FUNCTION_BLOCK L2_MedidorTapa_SFC EXTENDS L1_ControllerBase_SFC

VAR_INPUT 							// Sensores y comandos
	dh					: UINT; 	// Detector valor altura 
	// Lectura_Registrada	: BOOL;		// La lectura de la altura ha terminado 	
END_VAR

VAR_OUTPUT							// Actuadores
	L_1: BOOL; 						// Medidor de altura baja
	Leyendo: BOOL;
END_VAR

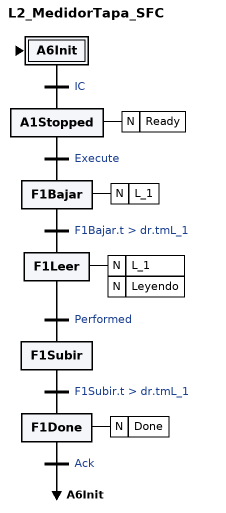
INITIAL_STEP A6Init:
END_STEP
TRANSITION FROM A6Init TO A1Stopped
    := IC;
END_TRANSITION
STEP A1Stopped:
    Ready(N);
END_STEP
TRANSITION FROM A1Stopped TO F1Bajar
    := Execute;
END_TRANSITION
STEP F1Bajar:
    L_1(N);
END_STEP
TRANSITION FROM F1Bajar TO F1Leer
    := F1Bajar.t > dr.tmL_1;
END_TRANSITION
STEP F1Leer:
    L_1(N);
    Leyendo(N);
END_STEP
TRANSITION FROM F1Leer TO F1Subir
    := Performed;
END_TRANSITION
STEP F1Subir:
END_STEP
TRANSITION FROM F1Subir TO F1Done
    := F1Subir.t > dr.tmL_1;
END_TRANSITION
STEP F1Done:
    Done(N);
END_STEP
TRANSITION FROM F1Done TO A6Init
    := Ack;
END_TRANSITION

END_FUNCTION_BLOCK

(* stored: Version 1.1.0.1, ProductVersion 3.1.4024.11
   POU L2_MedidorTapa_SFC: Id {586537d7-6cab-450b-b2b9-fb1352203f2f}, SpecialFunc None *)
